{attribute 'qualified_only'}
TYPE E_OpMod_AC :
(
	Invalid			:= 0,
	
	eOff			:= 1,
	eOn				:= 2,
	eNightCool		:= 3,
	eDisturb		:= 4,
	eSmokeExtract	:= 5,
	eFrost			:= 6,
	eFire			:= 7,
	eCentralOff		:= 8
	
) UDINT;
END_TYPE

(* stored: Version 1.1.0.1, ProductVersion 3.1.4024.5
   DUT E_OpMod_AC: Id {7c71ed4a-6636-4579-9333-127f74d2f93a} *)
